Staubli VAL3: countBool3D.pgx

public program countBool3D(bool& x_bInput[] (dimensions=3), num& x_nResult)
  local num l_nElement
  local num l_nDim[3]
begin

  x_nResult = 0

  for l_nDim[0] = 0 to size(x_bInput,1)-1
    for l_nDim[1] = 0 to size(x_bInput,2)-1
      for l_nDim[2] = 0 to size(x_bInput,3)-1
        if x_bInput[l_nDim[0], l_nDim[1], l_nDim[2]] == true
          x_nResult = x_nResult+1
        endIf
      endFor
    endFor
  endFor

end
